TYPE Jog_FxB_Type :
STRUCT
	 H_Open:  BOOL;
 H_Open_S:  BOOL;
 H_Close:  BOOL;
 H_Close_S:  BOOL;

 H_Hold:  BOOL;
 H_Hold_S:  BOOL;

 V_Open:  BOOL;
 V_Open_S: BOOL;
 V_Close: BOOL;
 V_Close_S: BOOL;

 
END_STRUCT
END_TYPE

(* stored: Version 1.1.0.1, ProductVersion 3.1.4024.15
   DUT Jog_FxB_Type: Id {4dc8c9a2-7bff-4c6d-9a71-f74fc1c4e50e} *)
